// ---- VISUs/Panels/Visualization.TcVIS
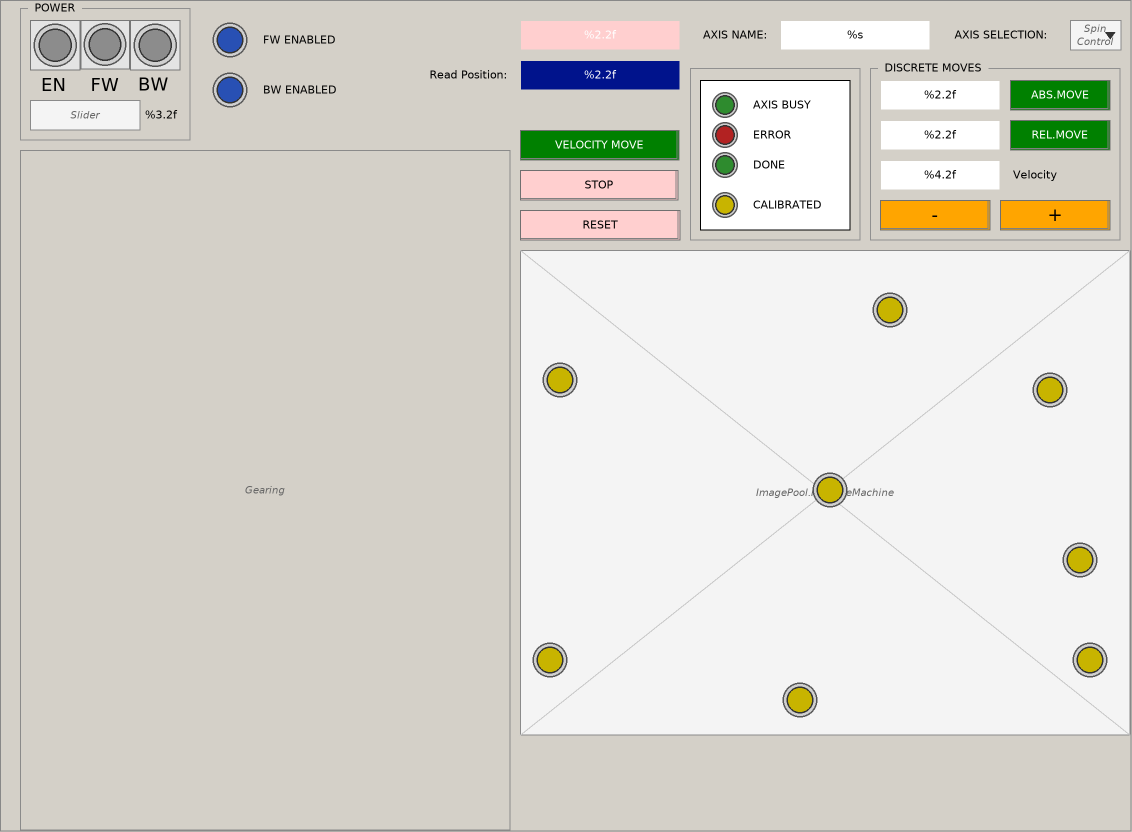
VISUALIZATION Visualization  // 1132x832
    GroupBox (870,60 250x180), "DISCRETE MOVES"
        Textfield (10,20 120x30), "%2.2f", text variable: GVL.axes[MAIN.hmiAxisSelect].fPosition
            OnMouseClick: write GVL.axes[MAIN.hmiAxisSelect].fPosition via Default
        Button (140,20 100x30), "ABS.MOVE", input disabled if: GVL.axes[MAIN.hmiAxisSelect].iAxisState=500
            OnMouseClick: execute { GVL.axes[MAIN.hmiAxisSelect].eCommand:=eMcCommand.MoveAbsolute; GVL.axes[MAIN.hmiAxisSelect].bEXECUTE:= TRUE; }
        Textfield (10,60 120x30), "%2.2f", text variable: GVL.axes[MAIN.hmiAxisSelect].fDistance
            OnMouseClick: write GVL.axes[MAIN.hmiAxisSelect].fDistance via Default
        Button (140,60 100x30), "REL.MOVE", input disabled if: GVL.axes[MAIN.hmiAxisSelect].iAxisState=500
            OnMouseClick: execute { GVL.axes[MAIN.hmiAxisSelect].eCommand:=eMcCommand.MoveRelative; GVL.axes[MAIN.hmiAxisSelect].bEXECUTE:= TRUE; }
        Button (10,140 110x30), "-"
            tap GVL.axes[MAIN.hmiAxisSelect].bJogBackward
            OnMouseClick: execute { GVL.axes[MAIN.hmiAxisSelect].eCommand:=eMcCommand.Jog; }
        Button (130,140 110x30), "+"
            tap GVL.axes[MAIN.hmiAxisSelect].bJogForward
            OnMouseClick: execute { GVL.axes[MAIN.hmiAxisSelect].eCommand:=eMcCommand.Jog; }
        Textfield (10,100 120x30), "%4.2f", text variable: GVL.axes[MAIN.hmiAxisSelect].fVelocity
            OnMouseClick: write GVL.axes[MAIN.hmiAxisSelect].fVelocity via Default
    Textfield (520,60 160x30), "%2.2f", text variable: GVL.axes[MAIN.hmiAxisSelect].Axis.NcToPlc.ActPos
    SpinControl (1070,20 51x30), variable: MAIN.hmiAxisSelect
        p651134158: GVL.axisNumMax
    Textfield (930,20 120x30), "AXIS SELECTION:", text variable: MAIN.hmiAxisSelect
    Textfield (1010,160 100x30), "Velocity", text variable: MAIN.hmiAxisSelect
    Textfield (650,20 120x30), "AXIS NAME:"
    GroupBox (20,0 170x140), "POWER"
        PushSwitchLed (110,20 50x50), variable: Limits.BwLimit[MAIN.hmiAxisSelect], behaviour: TOGGLE, style: Switch-PushSwitchLed-Gray
        Slider (10,100 110x30), variable: GVL.axes[MAIN.hmiAxisSelect].fOverride, scale 0..100
        Textfield (120,100 40x30), "%3.2f", text variable: GVL.axes[MAIN.hmiAxisSelect].fOverride
        Label (10,70 47x30), "EN"
        Label (110,70 47x29), "BW"
        PushSwitchLed (60,20 50x49), variable: Limits.FwLimit[MAIN.hmiAxisSelect], behaviour: TOGGLE, style: Switch-PushSwitchLed-Gray
        Label (60,70 50x30), "FW"
        PushSwitchLed (10,20 50x50), variable: GVL.axes[MAIN.hmiAxisSelect].bEnable, behaviour: TOGGLE, style: Switch-PushSwitchLed-Gray
    GroupBox (690,60 170x180)
        Rectangle (10,20 150x150)
        Lamp1 (20,30 30x30), variable: GVL.axes[MAIN.hmiAxisSelect].bBusy, style: Lamp-Lamp1-Green
        Lamp1 (20,60 30x30), variable: GVL.axes[MAIN.hmiAxisSelect].bError, style: Lamp-Lamp1-Red
        Lamp1 (20,90 30x30), variable: GVL.axes[MAIN.hmiAxisSelect].bDone, style: Lamp-Lamp1-Green
        Textfield (60,30 90x30), "AXIS BUSY", text variable: MAIN.hmiAxisSelect
        Textfield (60,60 90x30), "ERROR", text variable: MAIN.hmiAxisSelect
        Textfield (60,90 90x30), "DONE", text variable: MAIN.hmiAxisSelect
        Lamp1 (20,130 30x30), variable: GVL.axes[MAIN.hmiAxisSelect].Axis.Status.Homed, style: Lamp-Lamp1-Yellow
        Textfield (60,130 90x30), "CALIBRATED", text variable: MAIN.hmiAxisSelect
    Textfield (780,20 150x30), "%s", text variable: GVL.axes[MAIN.hmiAxisSelect].sAxisName
        OnMouseClick: write GVL.axes[MAIN.hmiAxisSelect].sAxisName via Edit
    Button (520,210 160x30), "RESET"
        OnMouseClick: execute { GVL.axes[MAIN.hmiAxisSelect].eCommand:=eMcCommand.Reset; GVL.axes[MAIN.hmiAxisSelect].bReset:= TRUE; }
    Image (520,250 610x485), image: ImagePool.NCStateMachine
    Lamp1 (1070,640 40x40), variable: GVL.axes[MAIN.hmiAxisSelect].iAxisState=100, style: Lamp-Lamp1-Yellow
    Lamp1 (780,680 40x40), variable: GVL.axes[MAIN.hmiAxisSelect].iAxisState=200, style: Lamp-Lamp1-Yellow
    Lamp1 (530,640 40x40), variable: GVL.axes[MAIN.hmiAxisSelect].iAxisState=300, style: Lamp-Lamp1-Yellow
    Lamp1 (1060,540 40x40), variable: GVL.axes[MAIN.hmiAxisSelect].iAxisState=999, style: Lamp-Lamp1-Yellow
    Lamp1 (810,470 40x40), variable: GVL.axes[MAIN.hmiAxisSelect].iAxisState=700, style: Lamp-Lamp1-Yellow
    Lamp1 (1030,370 40x40), variable: GVL.axes[MAIN.hmiAxisSelect].iAxisState=600, style: Lamp-Lamp1-Yellow
    Lamp1 (540,360 40x40), variable: GVL.axes[MAIN.hmiAxisSelect].iAxisState=400, style: Lamp-Lamp1-Yellow
    Lamp1 (870,290 40x40), variable: GVL.axes[MAIN.hmiAxisSelect].iAxisState=500, style: Lamp-Lamp1-Yellow
    TabControl (20,150 490x680)
        shows Gearing()
        shows Parameters()
        shows Homing()
        shows AxisSimulation()
        [0]: TabTitle=Gearing
        [1]: TabTitle=Parameters
        [2]: TabTitle=Adv. Homing
        [3]: TabTitle=Simulation
    Textfield (390,60 120x30), "Read Position:"
    Lamp1 (210,20 40x40), variable: GVL.axes[MAIN.hmiAxisSelect].bFwEnabled, style: Lamp-Lamp1-Blue
    Lamp1 (210,70 40x40), variable: GVL.axes[MAIN.hmiAxisSelect].bBwEnabled, style: Lamp-Lamp1-Blue
    Textfield (260,70 120x40), "BW ENABLED", text variable: MAIN.hmiAxisSelect
    Textfield (260,20 120x40), "FW ENABLED", text variable: MAIN.hmiAxisSelect
    Button (520,130 159x30), "VELOCITY MOVE", input disabled if: GVL.axes[MAIN.hmiAxisSelect].iAxisState=500
        OnMouseClick: execute { GVL.axes[MAIN.hmiAxisSelect].eCommand:=eMcCommand.MoveVelocity; GVL.axes[MAIN.hmiAxisSelect].bEXECUTE:= TRUE; }
    Button (520,170 158x30), "STOP"
        OnMouseClick: execute { GVL.axes[MAIN.hmiAxisSelect].eCommand:=eMcCommand.Stop; GVL.axes[MAIN.hmiAxisSelect].bExecute:= TRUE; }
    Textfield (520,20 160x30), "%2.2f", text variable: GVL.axes[MAIN.hmiAxisSelect].iErrorID
END_VISUALIZATION
